FUNCTION_BLOCK FB_TwoPositionPopIn
VAR_INPUT
	RepRate : BOOL; // TRUE - above RepRate Threshold
	Retracted_Pos1_IN :BOOL;
	Inserted_Pos2_IN : BOOL;
END_VAR
	
VAR_OUTPUT
	Insert_Pos2_OUT : BOOL;
	Interlock : BOOL; // MPS shutter
	State : E_2PosMonState;
	Error : BOOL; // timer expired
END_VAR

//Map the inputs to enum
IF Inserted_Pos2_IN AND Retracted_Pos1_IN THEN
	State:=E_2PosMonState.isBroken;
ELSIF Inserted_Pos2_IN AND NOT Retracted_Pos1_IN THEN
	State:=E_2PosMonState.isInserted;
ELSIF NOT Inserted_Pos2_IN AND Retracted_Pos1_IN THEN
	State:=E_2PosMonState.isRetracted;
ELSIF NOT Inserted_Pos2_IN AND NOT Retracted_Pos1_IN THEN
	State:=E_2PosMonState.isMoving;
END_IF


//Shutter interlock behaviour
IF State = E_2PosMonState.isBroken THEN //Broken
	Interlock := FALSE;
ELSIF State = E_2PosMonState.isMoving THEN //Moving
	Interlock := FALSE;
ELSIF State = E_2PosMonState.isInserted AND RepRate THEN
	Interlock := FALSE;	
ELSE 
	Interlock := TRUE;	
END_IF


// Air solenoid behaviour
IF RepRate THEN
	Retract();
	State := E_2PosMonState.isForcedOut;
END_IF

METHOD Control : BOOL
VAR_IN_OUT
	structure: ST_TwoPositionPopIn;
END_VAR

VAR
END_VAR
IF structure.InsertPos2Cmd THEN
	structure.InsertPos2Cmd := FALSE;
	Insert();	
END_IF


IF structure.RetractPos1Cmd THEN
	structure.RetractPos1Cmd := FALSE;
	Retract();	
END_IF

structure.StateSt := State;

structure.InsertedPos2St:=Inserted_Pos2_IN;
structure.RetractedPos1St:=Retracted_Pos1_IN;

structure.InterlockSt:=Interlock;
END_METHOD

METHOD Insert : BOOL
VAR_INPUT
END_VAR
IF RepRate THEN
	RETURN;
END_IF

Insert_Pos2_OUT := TRUE;
END_METHOD

METHOD Retract : BOOL
VAR_INPUT
END_VAR
Insert_Pos2_OUT := FALSE;
END_METHOD

END_FUNCTION_BLOCK

(* stored: Version 1.1.0.1, ProductVersion 3.1.4024.12
   POU FB_TwoPositionPopIn: Id {9e4b88f4-9d6f-4a56-97df-c904e208c07a}, SpecialFunc None
   Method Control: Id {76e1e668-265e-40f9-9c2f-c94d784ab45b}
   Method Insert: Id {6b27388e-dc96-4819-95a7-068dca6e0e24}
   Method Retract: Id {35ab9696-0cb4-4f7b-9473-5cef272e1475} *)
